Fanuc KAREL source: kt00536.KL

-- PROVISIONAL review KL for V940-1; original PC SHA256 bab827a71558bc8eeb0a8eca9e648bc170ba5cc7c4199721936a73a591435e76
-- Incomplete behavior may be omitted. Consult companion uncertainty JSON. Do not deploy.
PROGRAM KT00536
%NOLOCKGROUP
-- UNRESOLVED_DECL P1 type=000199
-- UNRESOLVED_DECL P2 type=000101
-- UNRESOLVED_DECL OUT type=000106
BEGIN
  -- V9_ZERO_TABLE_METADATA_HINT layout=0001; no indexed target words; source/name/runtime held
  -- UNRESOLVED_PC offsets 5-39; opcodes 49,7E,49,60,7E,4A
  -- UNRESOLVED_PC offsets 44-48; opcodes 7F
END KT00536
